TYPE ST_ModuleDataStatus :
STRUCT
	PublishedCount : UINT;
	Overflow : BOOL;
	DuplicateId : UDINT;
END_STRUCT
END_TYPE

(* stored: Version 1.1.0.1, ProductVersion 3.1.4026.18
   DUT ST_ModuleDataStatus: Id {e3273b41-d9ca-4b5a-9651-aea2757fc61a} *)
